SUBAPPLICATION Blink_LED (* Subapplication Type *)
  (* Standard: 61499-2 *)
  (* Version 1.0, 2023-10-23, franz *)
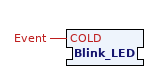
  EVENT_INPUT
    COLD;
  END_EVENT
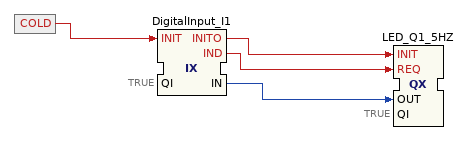
  FBS
    LED_Q1_5HZ : QX(QI := TRUE);
    DigitalInput_I1 : IX(QI := TRUE);
  END_FBS
  EVENT_CONNECTIONS
    COLD TO DigitalInput_I1.INIT;
    DigitalInput_I1.INITO TO LED_Q1_5HZ.INIT;
    DigitalInput_I1.IND TO LED_Q1_5HZ.REQ;
  END_CONNECTIONS
  DATA_CONNECTIONS
    DigitalInput_I1.IN TO LED_Q1_5HZ.OUT;
  END_CONNECTIONS
END_SUBAPPLICATION
